// TIA Portal V17 export
// export: Created 2023-03-06T02:05:26.1322136Z, ExportSetting WithDefaults, DisplayName Totally Integrated Automation Portal, DisplayVersion V17 Update 4, DisplayName TIA Portal Openness, DisplayVersion V17 Update 4, DisplayName TIA Portal Version Control Interface, DisplayVersion V17, DisplayName STEP 7 Professional, DisplayVersion V17 Update 4, DisplayName STEP 7 Safety, DisplayVersion V17, DisplayName WinCC Professional, DisplayVersion V17 Update 4
TYPE "BMS_TMS"
// stored: IsFailsafeCompliant false
   STRUCT
      xPwrOffCmd : Bool;   // TMS_Mode_Command = 0
      xCoolingCmd : Bool;   // TMS_Mode_Command = 1
      xHeatingCmd : Bool;   // TMS_Mode_Command = 2
      xSelfCircCmd : Bool;   // TMS_Mode_Command = 3
      iTempSet : Int;   // TMS_Value_Set_Temp
      xPwrOffSt : Bool;   // TMS_Real_Mode = 0
      xCoolingSt : Bool;   // TMS_Real_Mode = 1
      xHeatingSt : Bool;   // TMS_Real_Mode = 2
      xSelfCircSt : Bool;   // TMS_Real_Mode = 3
      rPowerMeas : Real;   // TMS_Demand_Power
      wCodeFlt : Word;   // TMS_Fault_Code
   END_STRUCT;
END_TYPE
